FUNCTION_BLOCK TwoConCtlMultiCast (* Composite Function Block Type *)
  (* Standard: 61499-2 *)
  (* Version 0.2, 2003-12-05, JHC, Rockwell Automation, Renamed from NEWCOMPFB. *)
  (* Version 0.1, 2002-01-08, JHC, Rockwell Automation, Added DLY FB as example. *)
  (* Version 0.0, 2000-05-27, JHC, Rockwell Automation *)
  (* Compiler header: package fb.rt.cs725; *)
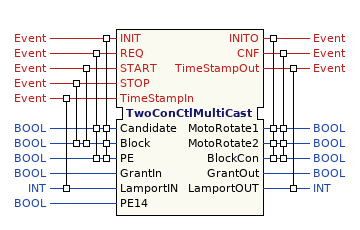
  EVENT_INPUT
    INIT WITH Candidate, Block, PE; (* Initialization Request *)
    REQ WITH Candidate, PE; (* Normal Execution Request *)
    START WITH Block;
    STOP WITH Block;
    TimeStampIn WITH LamportIN;
  END_EVENT
  EVENT_OUTPUT
    INITO WITH MotoRotate1, MotoRotate2, BlockCon; (* Initialization Confirm *)
    CNF WITH MotoRotate1, MotoRotate2, BlockCon; (* Execution Confirmation *)
    TimeStampOut WITH LamportOUT;
  END_EVENT
  VAR_INPUT
    Candidate : BOOL;
    Block : BOOL;
    PE : BOOL;
    GrantIn : BOOL;
    LamportIN : INT;
    PE14 : BOOL;
  END_VAR
  VAR_OUTPUT
    MotoRotate1 : BOOL;
    MotoRotate2 : BOOL;
    BlockCon : BOOL;
    GrantOut : BOOL;
    LamportOUT : INT;
  END_VAR
  FBS
    FC11 : ConveyorCTL(PE := 0, Block := 0, Candidate := 0);
    FC12 : ConveyorCTLMultiCast(ID := 1);
  END_FBS
  EVENT_CONNECTIONS
    INIT TO FC11.INIT;
    REQ TO FC11.REQ;
    FC12.INITO TO INITO;
    FC12.CNF TO CNF;
    REQ TO FC12.REQ;
    STOP TO FC12.CAS_STOP;
    START TO FC12.CAS_START;
    FC12.STOP TO FC11.CAS_STOP;
    FC12.START TO FC11.CAS_START;
    FC11.INITO TO FC12.INIT;
    TimeStampIn TO FC12.TimeStampIn;
    FC12.TimeStampOut TO TimeStampOut;
  END_CONNECTIONS
  DATA_CONNECTIONS
    Block TO FC12.Block;
    Candidate TO FC12.Candidate;
    PE TO FC12.PE;
    FC12.BlockCon TO BlockCon;
    FC11.MotoRotate TO MotoRotate1;
    FC12.MotoRotate TO MotoRotate2;
    PE14 TO FC12.PE14;
    GrantIn TO FC12.GrantIn;
    FC12.GrantOut TO GrantOut;
    FC12.LamportOUT TO LamportOUT;
    LamportIN TO FC12.LamportIN;
  END_CONNECTIONS
END_FUNCTION_BLOCK
